# EPICS substitutions: opcpaepsApp/Db/eps_leak_monitor.substitutions
file eps_leak_monitor.template {
  pattern
    {ID}
    {"01"}
    {"02"}
    {"03"}
    {"04"}
    {"05"}
    {"06"}
}
